FUNCTION RANGE_TO_WORD : WORD
VAR_INPUT
	X : REAL;
	low : REAL;
	high : REAL;
END_VAR


(*
version 1.0	9. jan 2008
programmer 	hugo
tested by		tobias

Range_to_word converts a real value between low and high into a byte

*)

RANGE_TO_WORD := DINT_TO_WORD(TRUNC_INT((LIMIT(low,X,high)-low) * 65535.0 / (high - low)));


(* revision history
hm	9. jan 2008		rev 1.0
	original version

*)

END_FUNCTION

(* stored: Version 1.1.0.1, ProductVersion 3.1.4022.7
   POU RANGE_TO_WORD: Id {5bb7e912-2005-49b0-9511-e16e808948c4}, SpecialFunc None *)
